{attribute 'qualified_only'}
{attribute 'strict'}
TYPE PackMLState :
(
	Aborting := 0,
	Aborted := 1,
	Clearing := 2,
	Stopping := 3,
	Stopped := 4,
	Resetting := 5,
	Idle := 6,
	Starting := 7,
	Execute := 8
);
END_TYPE

(* stored: Version 1.1.0.1, ProductVersion 3.1.4024.9
   DUT PackMLState: Id {cdcfd89e-3664-42f8-ab77-e96f8f186908} *)
